TYPE E_DisconnectorControlMode :
(
    MANUAL := 0,     // Manuel kontrol - Lokal butonlar
    AUTO := 1,       // Otomatik kontrol - PLC lojiği
    REMOTE := 2      // Uzaktan kontrol - SCADA/HMI
);
END_TYPE

(* stored: Version 1.1.0.1, ProductVersion 3.1.4024.15
   EnumerationTextList E_DisconnectorControlMode: Id {bff2dc10-0dd9-4cdf-8369-1c74838912d3} *)
